// TIA Portal V16 export
// export: Created 2021-11-12T13:32:14.7287619Z, ExportSetting WithDefaults, DisplayName Totally Integrated Automation Portal, DisplayVersion V16 Update 3, DisplayName TIA Portal Version Control Interface, DisplayVersion V16 Update 2, DisplayName TIA Portal Openness, DisplayVersion V16 Update 3, DisplayName SINAMICS Startdrive Advanced, DisplayVersion V16 Update 5, DisplayName SINAMICS Startdrive G130, G150, S120, S150, SINAMICS MV, S210, DisplayVersion V16 Update 5, DisplayName SINAMICS Startdrive G110M, G120, G120C, G120D, G120P, G115D, DisplayVersion V16 Update 5, DisplayName STEP 7 Professional, DisplayVersion V16 Update 3, DisplayName STEP 7 Safety, DisplayVersion V16, DisplayName WinCC UA Professional, DisplayVersion V16 Update 3
DATA_BLOCK "HMI_CMD_120"   // DB208
{ S7_Optimized_Access := 'TRUE' }
VERSION : 0.1
// stored: AutoNumber true, DBAccessibleFromOPCUA true, IsOnlyStoredInLoadMemory false, IsRetainMemResEnabled false, IsWriteProtectedInAS false, MemoryReserve 100
   VAR
      xxxxx___BinaryOthers___xxxxx : Byte;
      UH31_TA01_Ref { S7_SetPoint := 'True'} : Bool;   // Aligner - go to reference position
      WaitForNextPart : Bool := true;   // Conveyor - wait for next part from saw
      "UH31-FC01" { S7_SetPoint := 'True'} : "UDT_CH_DI_Command";   // Servoměnič TA01 je OK
      UC10_FC21 : "UDT_CH_DI_Command";   // 230V Part align OK
      UC12_FC01 : "UDT_CH_DI_Command";   // 400V Conveyor OK
      SF01_14 { S7_SetPoint := 'True'} : "UDT_CH_DI_Command";   // Conveyor Remote
      SF01_24 { S7_SetPoint := 'True'} : "UDT_CH_DI_Command";   // Conveyor Automat
      SF03_14 { S7_SetPoint := 'True'} : "UDT_CH_DI_Command";   // Conveyor Start Automat
      SF04_12 { S7_SetPoint := 'True'} : "UDT_CH_DI_Command";   // Conveyor Stop
      SF05_14 { S7_SetPoint := 'True'} : "UDT_CH_DI_Command";   // Conveyor Manual backwards
      SF05_24 { S7_SetPoint := 'True'} : "UDT_CH_DI_Command";   // Conveyor Manual forward
      SF06_14 { S7_SetPoint := 'True'} : "UDT_CH_DI_Command";   // Conveyor lift 1 up
      SF06_24 { S7_SetPoint := 'True'} : "UDT_CH_DI_Command";   // Conveyor lift 1 down
      SF07_14 { S7_SetPoint := 'True'} : "UDT_CH_DI_Command";   // Conveyor lift 2 up
      SF07_24 { S7_SetPoint := 'True'} : "UDT_CH_DI_Command";   // Conveyor lift 2 down
      SF08_14 { S7_SetPoint := 'True'} : "UDT_CH_DI_Command";   // Conveyor lift 3 up
      SF08_24 { S7_SetPoint := 'True'} : "UDT_CH_DI_Command";   // Conveyor lift 3 down
      SF09_14 { S7_SetPoint := 'True'} : "UDT_CH_DI_Command";   // Conveyor lift 4 up
      SF09_24 { S7_SetPoint := 'True'} : "UDT_CH_DI_Command";   // Conveyor lift 4 down
      SF10_14 { S7_SetPoint := 'True'} : "UDT_CH_DI_Command";   // Conveyor aligning align
      SF10_24 { S7_SetPoint := 'True'} : "UDT_CH_DI_Command";   // Conveyor aligning release
      SF11_14 { S7_SetPoint := 'True'} : "UDT_CH_DI_Command";   // Conveyor Stopper up
      SF11_24 { S7_SetPoint := 'True'} : "UDT_CH_DI_Command";   // Conveyor Stopper down
      xxxxx___BinarySensors___xxxxx : Byte;
      GL01_BG01 : "UDT_CH_DI_Command";   // Proximitní senzor - Koncák pro referenci
      GL01_BG01R : "UDT_CH_DI_Command";   // Proximitní senzor - Zarážka nahoře
      GL01_BG01V : "UDT_CH_DI_Command";   // Proximitní senzor - Zarážka dole
      GL01_BG02 : "UDT_CH_DI_Command";   // Optický senzor - Přítomnost přířezu v pozici po vykulení
      GM01_BG01R : "UDT_CH_DI_Command";   // Indukční senzor - Výtah 1 dole
      GM01_BG01V : "UDT_CH_DI_Command";   // Indukční senzor - Výtah 1 nahoře
      GM01_BG02R : "UDT_CH_DI_Command";   // Indukční senzor - Výtah 2 dole
      GM01_BG02V : "UDT_CH_DI_Command";   // Indukční senzor - Výtah 2 nahoře
      GM01_BG03R : "UDT_CH_DI_Command";   // Indukční senzor - Výtah 3 dole
      GM01_BG03V : "UDT_CH_DI_Command";   // Indukční senzor - Výtah 3 nahoře
      GM01_BG04R : "UDT_CH_DI_Command";   // Indukční senzor - Výtah 4 dole
      GM01_BG04V : "UDT_CH_DI_Command";   // Indukční senzor - Výtah 4 nahoře
      GL01_BG03 : "UDT_CH_DI_Command";   // Optický senzor - Přířez na řetěze před výtahama
      GM01_BG01 : "UDT_CH_DI_Command";   // Optický senzor - Přířez na řetěze výtah 1
      GM01_BG02 : "UDT_CH_DI_Command";   // Optický senzor - Přířez na řetěze výtah 2
      GM01_BG03 : "UDT_CH_DI_Command";   // Optický senzor - Přířez na řetěze výtah 3
      GM01_BG04 : "UDT_CH_DI_Command";   // Optický senzor - Přířez na řetěze výtah 4
      GL01_BG04 : "UDT_CH_DI_Command";   // Optický senzor - Přířez na řetěze výtah 5
      GL01_BG5 : "UDT_CH_DI_Command";   // Enkodér na dopravníku
      xxxxx___Drives___xxxxx : Byte;
      GL01_MA01 : "UDT_Drive1_Command";   // Dorážení přířezu ke kraji
      GL01_MA02 : "UDT_Drive1_Command";   // Pohon dopravníku
      UC12_TA01 : "UDT_SINAMICS_G120_Command";   // Měnič
      GL01_BG05 { S7_SetPoint := 'True'} : "UDT_MCEnkoder_Command";   // Enkodér
      UH31_TA01 : "UDT_FESTO_CMMT_Command";   // Řízení servomotoru - FESTO
      xxxxx___Valves___xxxxx : Byte;
      GL01_MM01 : "UDT_Valve2WB_Command";   // Pneumatický válec - Zarážka pro vykulení
      GM01_MM01 : "UDT_Valve2WB_Command";   // Pneumatický válec - Zvedání přířezu - Výtah 1
      GM01_MM02 : "UDT_Valve2WB_Command";   // Pneumatický válec - Zvedání přířezu - Výtah 2
      GM01_MM03 : "UDT_Valve2WB_Command";   // Pneumatický válec - Zvedání přířezu - Výtah 3
      GM01_MM04 : "UDT_Valve2WB_Command";   // Pneumatický válec - Zvedání přířezu - Výtah 4
      xxxxx__MaterialFlow__xxxxx : Byte;
      MatCard : "UDT_MatCard_Cmd";   // Material flow commands
      xxxxx___SensorsAlarms___xxxxx { S7_SetPoint := 'True'} : Byte;
      GL01_MM01_Alarm { S7_SetPoint := 'True'} : "UDT_DI_Mon_Command";   // Stopper discrepance senzorů
      GM01_MM01_Alarm { S7_SetPoint := 'True'} : "UDT_DI_Mon_Command";   // Výtah 1 - discrepance senzorů
      GM01_MM02_Alarm { S7_SetPoint := 'True'} : "UDT_DI_Mon_Command";   // Výtah 2 - discrepance senzorů
      GM01_MM03_Alarm { S7_SetPoint := 'True'} : "UDT_DI_Mon_Command";   // Výtah 3 - discrepance senzorů
      GM01_MM04_Alarm { S7_SetPoint := 'True'} : "UDT_DI_Mon_Command";   // Výtah 4 - discrepance senzorů
      xxxxx___ProcessAlarms___xxxxx : Byte;
      DataTracking_1 : "UDT_DI_Mon_Command";   // part in stopping position not on map
      DataTracking_2 { S7_SetPoint := 'True'} : "UDT_DI_Mon_Command";   // part in lift 1 position not on map
      DataTracking_3 { S7_SetPoint := 'True'} : "UDT_DI_Mon_Command";   // part in lift 2 position not on map
      DataTracking_4 { S7_SetPoint := 'True'} : "UDT_DI_Mon_Command";   // part in lift 3 position not on map
      DataTracking_5 { S7_SetPoint := 'True'} : "UDT_DI_Mon_Command";   // part in lift 4 position not on map
      DataTracking_6 { S7_SetPoint := 'True'} : "UDT_DI_Mon_Command";   // part in before lifts position not on map
      Senzor_1 : "UDT_DI_Mon_Command";   // part in stopping position not on senzor
      Senzor_2 { S7_SetPoint := 'True'} : "UDT_DI_Mon_Command";   // part in lift 1 position not on senzor
      Senzor_3 { S7_SetPoint := 'True'} : "UDT_DI_Mon_Command";   // part in lift 2 position not on senzor
      Senzor_4 { S7_SetPoint := 'True'} : "UDT_DI_Mon_Command";   // part in lift 3 position not on senzor
      Senzor_5 { S7_SetPoint := 'True'} : "UDT_DI_Mon_Command";   // part in lift 4 position not on senzor
      Senzor_6 { S7_SetPoint := 'True'} : "UDT_DI_Mon_Command";   // part in before lifts position not on senzor
      UC10_FC21_Alarm { S7_SetPoint := 'True'} : "UDT_DI_Mon_Command";   // 230V Part align NOK
      UC12_FC01_Alarm { S7_SetPoint := 'True'} : "UDT_DI_Mon_Command";   // 400V Conveyor NOK
      ConvOverflow { S7_SetPoint := 'True'} : "UDT_DI_Mon_Command";   // part behind last lift
      ConvStepTooLong { S7_SetPoint := 'True'} : "UDT_DI_Mon_Command";   // conveyor step is too long
   END_VAR
BEGIN
END_DATA_BLOCK
